// TIA Portal V16 export
// export: Created 2022-02-28T20:45:45.7558179Z, ExportSetting WithDefaults, DisplayName Totally Integrated Automation Portal, DisplayVersion V16, DisplayName TIA Portal Version Control Interface, DisplayVersion V16, DisplayName TIA Portal Openness, DisplayVersion V16, DisplayName STEP 7 Professional, DisplayVersion V16, DisplayName STEP 7 Safety, DisplayVersion V16, DisplayName WinCC Advanced, DisplayVersion V16
DATA_BLOCK "01_PLC-Software"   // DB1
{ S7_Optimized_Access := 'TRUE' }
VERSION : 0.1
// stored: AutoNumber true, DBAccessibleFromOPCUA true, IsOnlyStoredInLoadMemory false, IsRetainMemResEnabled false, IsWriteProtectedInAS false, MemoryReserve 100
   VAR
      IN_Pistilos : Array[0..14] of Bool;
      IN_Pentoflex : Array[0..14] of Bool;
      IN_Cam_Pistilos : Array[0..14] of Bool;
      IN_Cam_Pentoflex : Array[0..14] of Bool;
      OUT_Pistilos : Array[0..7] of Bool;
      OUT_Pentoflex : Array[0..7] of Bool;
      Pistilos_Estados_Varidor : Array[0..7] of Bool;
      Alarmas : Array[0..14] of Int;
      Estado_Proceso : Array[0..14] of Bool;
   END_VAR
BEGIN
   // IN_Pistilos[0] : Paro Emerg Pistilos
   // IN_Pistilos[1] : Start Pistilos
   // IN_Pistilos[2] : Stop Pistilos
   // IN_Pistilos[3] : Trigger Cam 1
   // IN_Pentoflex[0] : Paro Emerg Producto Final
   // IN_Pentoflex[1] : Start Producto Final
   // IN_Pentoflex[2] : Stop Producto Final
   // IN_Pentoflex[3] : Trigger Cam 2 Final
   // OUT_Pistilos[0] : Motor Pistilos
   // OUT_Pentoflex[0] : Motor Pentoflex
   // Pistilos_Estados_Varidor[0] : Variador 1 ok
   // Alarmas[0] : Alarma PE Pistilos
   // Alarmas[1] : Alarma_Fallo_Cam_Pistilos
   // Alarmas[2] : Alarma_NLectura_Cam_Pistilos
   // Alarmas[3] : Alarma_NCoincidencia_Cam_Pistilos
   // Alarmas[4] : Alama PE Pentoflex
   // Alarmas[5] : Alarma_Fallo_Cam_Pentoflex
   // Alarmas[6] : Alarma_NLectura_Cam_Pentoflex
   // Alarmas[7] : Alarma_NCoincidencia_Cam_Pentoflex
   // Estado_Proceso[0] : Arranque Modo Automático Pistilos
   // Estado_Proceso[1] : Arranque Modo Manual Pistilos
   // Estado_Proceso[2] : Arranque Modo Automático Pentoflex
   // Estado_Proceso[3] : Arranque Modo Manual Pentoflex
END_DATA_BLOCK
